# EPICS autosave request: iocBoot/generic_motors_ioc/dbSave/HS_Ah_.req
%
% BURT Request File
%
% $(P)HS:Ah:  Huber slits, Horizontal Aperture
%

file assy.req ASSY=$(P)HS:Ah
$(P)HS:Ah:Invert
file mtr1.req MTR1=$(P)HS:mo
file mtr1.req MTR1=$(P)HS:mi
file drv1.req DRV1=$(P)HS:YO
file drv1.req DRV1=$(P)HS:YI
file axs1.req AXS1=$(P)HS:YC
file axs1.req AXS1=$(P)HS:YS
